// TIA Portal V16 export
// export: Created 2022-11-17T15:49:50.8751186Z, ExportSetting WithDefaults, DisplayName Totally Integrated Automation Portal, DisplayVersion V16 Update 6, DisplayName TIA Portal Version Control Interface, DisplayVersion V16 Update 2, DisplayName TIA Portal Openness, DisplayVersion V16 Update 6, DisplayName SINAMICS Startdrive Advanced, DisplayVersion V16 Update 5, DisplayName SINAMICS Startdrive G130, G150, S120, S150, SINAMICS MV, S210, DisplayVersion V16 Update 5, DisplayName SINAMICS Startdrive G110M, G120, G120C, G120D, G120P, G115D, DisplayVersion V16 Update 5, DisplayName STEP 7 Professional, DisplayVersion V16 Update 6, DisplayName STEP 7 Safety, DisplayVersion V16, DisplayName WinCC Advanced, DisplayVersion V16 Update 6
TYPE "APP"
// stored: IsFailsafeCompliant false
   STRUCT
      PID_ComponenteProporzionale : DInt;
      PID_ComponenteIntegrale : DInt;
      PID_ComponenteDerivativa : DInt;
      Tiro : Int;   // Valore di tiro richiesto: 1-100 => 1-100% Setup 1, 101-200 => 1-100% Setup 2, 0 => Azzera regolatore
      Tiro1 : Int;
      Tiro2 : Int;
      TiroPrecedente : Int;   // Valore di tiro richiesto istante (n-1)
      TiroAppoggio : Int;
      ErroreAttuale : Int;   // Errore istante (n)
      ErrorePrecedente : Int;   // Errore istante (n-1)
      PID_Kp : Int;   // Kp in uso nel PID
      PID_Ki : Int;   // Ki in uso nel PID
      PID_Kd : Int;   // Kd in uso nel PID
      SetpointTiro : Int;   // Valore di setpoint del PID
      SetpointTiroRampa : Int;   // Valore di setpoint del PID iniziale a rampa
      TransitorioInizialeFase1 : Int;   // Indica che si deve eseguire la rampa iniziale (Fase 1)
      TransitorioFase3 : Int;   // Indica che si deve eseguire la rampa da velocita' alta a media (Fase 3)
      TransitorioFase4 : Int;   // Indica che si deve eseguire la rampa da velocita' media a bassa (Fase 4)
      VelocitaRotazione : Int;   // Velocita' di rotazione richiesta
      VelocitaRotazioneFase2 : Int;   // Velocita' di rotazione richiesta durante la Fase 2
      VelocitaRotazioneAppoggio1 : Int;
      VelocitaRotazioneAppoggio2 : Int;
      Fase1OneShoot : Int;   // Indica che sono appena entrato nella fase di traansitorio di accelerazione (Fase 1)
      Fase2OneShoot : Int;   // Indica che sono appena entrato nella fase di transitorio iniziale (Fase 2)
      Fase3OneShoot : Int;   // Indica che sono appena entrato nella fase di transitorio di velocita' alta - media (Fase 3)
      Fase4OneShoot : Int;   // Indica che sono appena entrato nella fase di transitorio di velocita' media - bassa (Fase 4)
      ArrestoRepentinoOneShoot : Int;   // Indica che sono appena entrato nella fase di arresto repentino
      TiroFase1 : Int;   // Indica il tiro nella Fase 1 usato nella Fase 2
      TempIntero : Int;
      Fase : Int;
      BallerinoPrecedente : Array[0..2] of Int;   // Valore del ballerino negli istanti precedenti
      LimiteComponenteIntegrale : Int;   // Limite della componente integrale durante la transizione dalla velocita alta a media (Fase 3) e dalla media a bassa (Fase 4)
      TiroRichiesto : Int;   // Valore di tiro compreso fra 1 e 100 richiesto dalla logica di controllo
      TimerArrestoRepentino : Int;   // Timer per arresto repentino.
      TiroMinimoArrestoRepentino : Int;   // Tiro minimo durante un'arresto repentino
      VariazioneTiro : Int;   // Variazione del tiro film (ballerino)
      TimerFase2 : Int;   // Timer usato nella Fase 2 per arrestare i rulli in caso di rottura film
      TempoRotturaFilm : Int;   // Tempo rottura film in numero di scansioni (1 scansione ogni 30msec)
      TimerFase4 : Int;   // Timer per Fase 4
      TiroMinimoFase4 : Int;   // Tiro minimo durante la Fase 4 di arresto
      PID_Uscita : DInt;   // Valore di uscita del PID
      PrestiroRichiesto : DInt;   // Valore di prestiro richiesto. Valore compreso fra 0 e 500
      PrestiroAppoggio : Real;
   END_STRUCT;
END_TYPE
